// TIA Portal V17 export
// export: Created 2023-02-14T02:49:44.5105658Z, ExportSetting WithDefaults, DisplayName Totally Integrated Automation Portal, DisplayVersion V17, DisplayName TIA Portal Openness, DisplayVersion V17, DisplayName TIA Portal Teamcenter Gateway, DisplayVersion V17, DisplayName TIA Portal Version Control Interface, DisplayVersion V17, DisplayName SINAMICS Startdrive Advanced, DisplayVersion V17, DisplayName SINAMICS Startdrive G130, G150, S120, S150, SINAMICS MV, S210, DisplayVersion V17, DisplayName SINAMICS Startdrive G110M, G120, G120C, G120D, G120P, G115D, DisplayVersion V17, DisplayName STEP 7 Professional, DisplayVersion V17, DisplayName STEP 7 Safety, DisplayVersion V17, DisplayName WinCC Professional, DisplayVersion V17
FUNCTION_BLOCK "ReadDateandTime"   // FB31, LAD
{ S7_Optimized_Access := 'TRUE' }
VERSION : 0.1
// stored: AutoNumber false, IsIECCheckEnabled false, IsRetainMemResEnabled false, MemoryReserve 100, SetENOAutomatically false, UDAEnableTagReadback false
   VAR
      Rd_LocDTL : DTL;
      Rd_LocDTL_Retval : Int;
      LocDT_Out : Date_And_Time;
      LocDT_Retval : Int;
      LocLDT_Out : LDT;
      LocDLT_Retval : Int;
   END_VAR
BEGIN

REGION Network 1: Read Local Date and Time
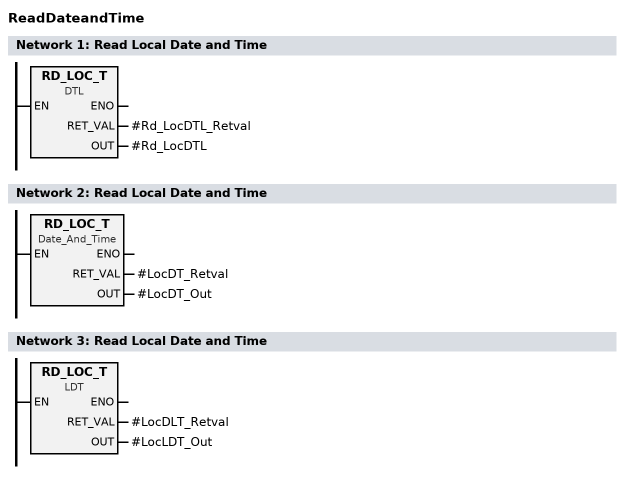
   RUNG wire#powerrail
      { S7_Templates := "date_type := DTL" } RD_LOC_T(RET_VAL => #Rd_LocDTL_Retval, OUT => #Rd_LocDTL)
   END_RUNG
   // the same network as SCL:
   #Rd_LocDTL_Retval := RD_LOC_T(OUT => #Rd_LocDTL);
END_REGION

REGION Network 2: Read Local Date and Time
   RUNG wire#powerrail
      { S7_Templates := "date_type := Date_And_Time" } RD_LOC_T(RET_VAL => #LocDT_Retval, OUT => #LocDT_Out)
   END_RUNG
   // the same network as SCL:
   #LocDT_Retval := RD_LOC_T(OUT => #LocDT_Out);
END_REGION

REGION Network 3: Read Local Date and Time
   RUNG wire#powerrail
      { S7_Templates := "date_type := LDT" } RD_LOC_T(RET_VAL => #LocDLT_Retval, OUT => #LocLDT_Out)
   END_RUNG
   // the same network as SCL:
   #LocDLT_Retval := RD_LOC_T(OUT => #LocLDT_Out);
END_REGION
END_FUNCTION_BLOCK
